// TIA Portal V16 export
// export: Created 2022-03-28T07:44:05.7115282Z, ExportSetting WithDefaults, DisplayName Totally Integrated Automation Portal, DisplayVersion V16 Update 5, DisplayName TIA Portal Version Control Interface, DisplayVersion V16 Update 2, DisplayName TIA Portal Openness, DisplayVersion V16 Update 5, DisplayName STEP 7 Professional, DisplayVersion V16 Update 5, DisplayName STEP 7 Safety, DisplayVersion V16, DisplayName WinCC Professional, DisplayVersion V16 Update 5
FUNCTION "fc_04_HMI" : Void   // FC4, LAD
{ S7_Optimized_Access := 'TRUE' }
VERSION : 0.1
// stored: AutoNumber false, IsIECCheckEnabled false, SetENOAutomatically false, UDAEnableTagReadback false
   VAR_TEMP   // added for the SCL form of the ladder/FBD networks
      _w1 : Bool;
      _w2 : Bool;
      _w3 : Bool;
   END_VAR
BEGIN

REGION Network 1
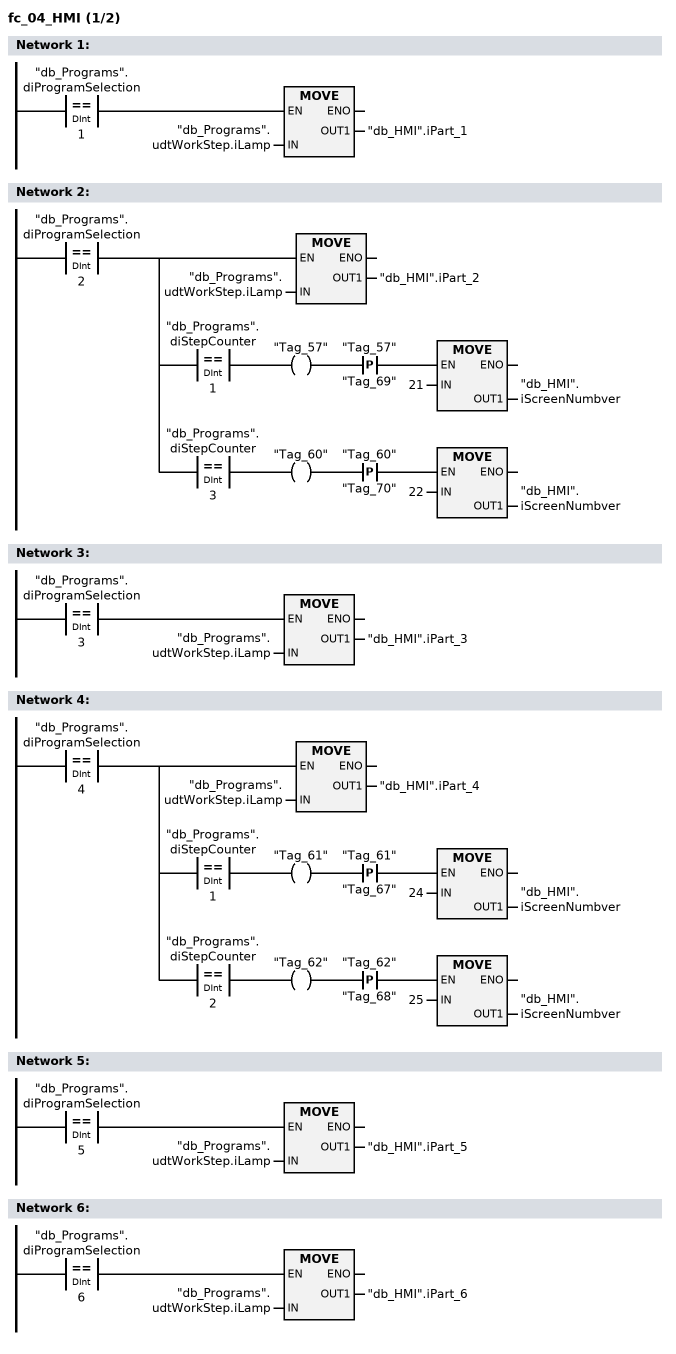
   RUNG wire#powerrail
      { S7_Templates := "SrcType := DInt" } EQ_Contact(in1 := "db_Programs".diProgramSelection, in2 := 1)
      Move(in := "db_Programs".udtWorkStep.iLamp, out1 => "db_HMI".iPart_1)
   END_RUNG
   // the same network as SCL:
   IF "db_Programs".diProgramSelection = 1 THEN "db_HMI".iPart_1 := "db_Programs".udtWorkStep.iLamp; END_IF;
END_REGION

REGION Network 2
   RUNG wire#powerrail
      { S7_Templates := "SrcType := DInt" } EQ_Contact(in1 := "db_Programs".diProgramSelection, in2 := 2)
      wire#w1
      Move(in := "db_Programs".udtWorkStep.iLamp, out1 => "db_HMI".iPart_2)
   END_RUNG
   RUNG wire#w1
      { S7_Templates := "SrcType := DInt" } EQ_Contact(in1 := "db_Programs".diStepCounter, in2 := 1)
      Coil( "Tag_57" )
      P_Contact(operand := "Tag_57", bit := "Tag_69")
      Move(in := 21, out1 => "db_HMI".iScreenNumbver)
   END_RUNG
   RUNG wire#w1
      { S7_Templates := "SrcType := DInt" } EQ_Contact(in1 := "db_Programs".diStepCounter, in2 := 3)
      Coil( "Tag_60" )
      P_Contact(operand := "Tag_60", bit := "Tag_70")
      Move(in := 22, out1 => "db_HMI".iScreenNumbver)
   END_RUNG
   // the same network as SCL:
   #_w1 := "db_Programs".diProgramSelection = 2;
   IF #_w1 THEN "db_HMI".iPart_2 := "db_Programs".udtWorkStep.iLamp; END_IF;
   "Tag_57" := #_w1 AND ("db_Programs".diStepCounter = 1);
   #_w2 := "Tag_57" AND "Tag_57" AND NOT "Tag_69";   // rising edge of "Tag_57"
   "Tag_69" := "Tag_57";
   IF #_w2 THEN "db_HMI".iScreenNumbver := 21; END_IF;
   "Tag_60" := #_w1 AND ("db_Programs".diStepCounter = 3);
   #_w3 := "Tag_60" AND "Tag_60" AND NOT "Tag_70";   // rising edge of "Tag_60"
   "Tag_70" := "Tag_60";
   IF #_w3 THEN "db_HMI".iScreenNumbver := 22; END_IF;
END_REGION

REGION Network 3
   RUNG wire#powerrail
      { S7_Templates := "SrcType := DInt" } EQ_Contact(in1 := "db_Programs".diProgramSelection, in2 := 3)
      Move(in := "db_Programs".udtWorkStep.iLamp, out1 => "db_HMI".iPart_3)
   END_RUNG
   // the same network as SCL:
   IF "db_Programs".diProgramSelection = 3 THEN "db_HMI".iPart_3 := "db_Programs".udtWorkStep.iLamp; END_IF;
END_REGION

REGION Network 4
   RUNG wire#powerrail
      { S7_Templates := "SrcType := DInt" } EQ_Contact(in1 := "db_Programs".diProgramSelection, in2 := 4)
      wire#w1
      Move(in := "db_Programs".udtWorkStep.iLamp, out1 => "db_HMI".iPart_4)
   END_RUNG
   RUNG wire#w1
      { S7_Templates := "SrcType := DInt" } EQ_Contact(in1 := "db_Programs".diStepCounter, in2 := 1)
      Coil( "Tag_61" )
      P_Contact(operand := "Tag_61", bit := "Tag_67")
      Move(in := 24, out1 => "db_HMI".iScreenNumbver)
   END_RUNG
   RUNG wire#w1
      { S7_Templates := "SrcType := DInt" } EQ_Contact(in1 := "db_Programs".diStepCounter, in2 := 2)
      Coil( "Tag_62" )
      P_Contact(operand := "Tag_62", bit := "Tag_68")
      Move(in := 25, out1 => "db_HMI".iScreenNumbver)
   END_RUNG
   // the same network as SCL:
   #_w1 := "db_Programs".diProgramSelection = 4;
   IF #_w1 THEN "db_HMI".iPart_4 := "db_Programs".udtWorkStep.iLamp; END_IF;
   "Tag_61" := #_w1 AND ("db_Programs".diStepCounter = 1);
   #_w2 := "Tag_61" AND "Tag_61" AND NOT "Tag_67";   // rising edge of "Tag_61"
   "Tag_67" := "Tag_61";
   IF #_w2 THEN "db_HMI".iScreenNumbver := 24; END_IF;
   "Tag_62" := #_w1 AND ("db_Programs".diStepCounter = 2);
   #_w3 := "Tag_62" AND "Tag_62" AND NOT "Tag_68";   // rising edge of "Tag_62"
   "Tag_68" := "Tag_62";
   IF #_w3 THEN "db_HMI".iScreenNumbver := 25; END_IF;
END_REGION

REGION Network 5
   RUNG wire#powerrail
      { S7_Templates := "SrcType := DInt" } EQ_Contact(in1 := "db_Programs".diProgramSelection, in2 := 5)
      Move(in := "db_Programs".udtWorkStep.iLamp, out1 => "db_HMI".iPart_5)
   END_RUNG
   // the same network as SCL:
   IF "db_Programs".diProgramSelection = 5 THEN "db_HMI".iPart_5 := "db_Programs".udtWorkStep.iLamp; END_IF;
END_REGION

REGION Network 6
   RUNG wire#powerrail
      { S7_Templates := "SrcType := DInt" } EQ_Contact(in1 := "db_Programs".diProgramSelection, in2 := 6)
      Move(in := "db_Programs".udtWorkStep.iLamp, out1 => "db_HMI".iPart_6)
   END_RUNG
   // the same network as SCL:
   IF "db_Programs".diProgramSelection = 6 THEN "db_HMI".iPart_6 := "db_Programs".udtWorkStep.iLamp; END_IF;
END_REGION

REGION Network 7
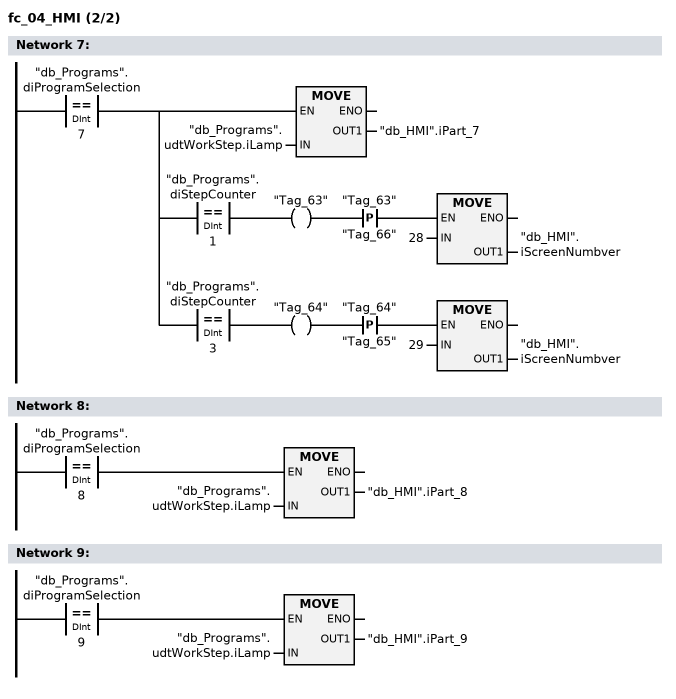
   RUNG wire#powerrail
      { S7_Templates := "SrcType := DInt" } EQ_Contact(in1 := "db_Programs".diProgramSelection, in2 := 7)
      wire#w1
      Move(in := "db_Programs".udtWorkStep.iLamp, out1 => "db_HMI".iPart_7)
   END_RUNG
   RUNG wire#w1
      { S7_Templates := "SrcType := DInt" } EQ_Contact(in1 := "db_Programs".diStepCounter, in2 := 1)
      Coil( "Tag_63" )
      P_Contact(operand := "Tag_63", bit := "Tag_66")
      Move(in := 28, out1 => "db_HMI".iScreenNumbver)
   END_RUNG
   RUNG wire#w1
      { S7_Templates := "SrcType := DInt" } EQ_Contact(in1 := "db_Programs".diStepCounter, in2 := 3)
      Coil( "Tag_64" )
      P_Contact(operand := "Tag_64", bit := "Tag_65")
      Move(in := 29, out1 => "db_HMI".iScreenNumbver)
   END_RUNG
   // the same network as SCL:
   #_w1 := "db_Programs".diProgramSelection = 7;
   IF #_w1 THEN "db_HMI".iPart_7 := "db_Programs".udtWorkStep.iLamp; END_IF;
   "Tag_63" := #_w1 AND ("db_Programs".diStepCounter = 1);
   #_w2 := "Tag_63" AND "Tag_63" AND NOT "Tag_66";   // rising edge of "Tag_63"
   "Tag_66" := "Tag_63";
   IF #_w2 THEN "db_HMI".iScreenNumbver := 28; END_IF;
   "Tag_64" := #_w1 AND ("db_Programs".diStepCounter = 3);
   #_w3 := "Tag_64" AND "Tag_64" AND NOT "Tag_65";   // rising edge of "Tag_64"
   "Tag_65" := "Tag_64";
   IF #_w3 THEN "db_HMI".iScreenNumbver := 29; END_IF;
END_REGION

REGION Network 8
   RUNG wire#powerrail
      { S7_Templates := "SrcType := DInt" } EQ_Contact(in1 := "db_Programs".diProgramSelection, in2 := 8)
      Move(in := "db_Programs".udtWorkStep.iLamp, out1 => "db_HMI".iPart_8)
   END_RUNG
   // the same network as SCL:
   IF "db_Programs".diProgramSelection = 8 THEN "db_HMI".iPart_8 := "db_Programs".udtWorkStep.iLamp; END_IF;
END_REGION

REGION Network 9
   RUNG wire#powerrail
      { S7_Templates := "SrcType := DInt" } EQ_Contact(in1 := "db_Programs".diProgramSelection, in2 := 9)
      Move(in := "db_Programs".udtWorkStep.iLamp, out1 => "db_HMI".iPart_9)
   END_RUNG
   // the same network as SCL:
   IF "db_Programs".diProgramSelection = 9 THEN "db_HMI".iPart_9 := "db_Programs".udtWorkStep.iLamp; END_IF;
END_REGION
END_FUNCTION
